KUKA KRL program: kukaSplineTemplate.src, kukaSplineTemplate.dat

--- kukaSplineTemplate.src ---
&ACCESS RVP
&REL 2
&PARAM EDITMASK = *
&PARAM TEMPLATE = C:\KRC\Roboter\Template\vorgabe
DEF mimi( )
;FOLD INI;%{PE}
  ;FOLD BASISTECH INI
    GLOBAL INTERRUPT DECL 3 WHEN $STOPMESS==TRUE DO IR_STOPM ( )
    INTERRUPT ON 3
    BAS (#INITMOV,0 )
  ;ENDFOLD (BASISTECH INI)
  ;FOLD USER INI
    ;Make your modifications here

  ;ENDFOLD (USER INI)
;ENDFOLD (INI)

;FOLD PTP HOME  Vel= 2 % DEFAULT;%{PE}%MKUKATPBASIS,%CMOVE,%VPTP,%P 1:PTP, 2:HOME, 3:, 5:100, 7:DEFAULT
$BWDSTART = FALSE
PDAT_ACT=PDEFAULT
FDAT_ACT=FHOME
BAS (#PTP_PARAMS,2 )
$H_POS=XHOME
PTP  XHOME
;ENDFOLD

$BWDSTART=FALSE
LDAT_ACT=LCPDAT[[firstIndex]]
FDAT_ACT=FP[[firstIndex]]
BAS(#CP_PARAMS,2)

;FOLD Shape SPLINE
	SPLINE
		TIME_BLOCK START
		[[range .Points]]
			SPL XP[[.Index]]
			[[if .TimeMark]]
			;Time mark at [[.TimeCode]]s with value [[.TimeMark]]s
			TIME_BLOCK PART = [[.TimeMark]]
			[[end]]
			[[if rMarkTest .Index .TimeMark]]
			;Time mark at [[.TimeCode]]s with value [[rTime]]s
			TIME_BLOCK PART = [[rTime]]
			[[end]]
		[[end]]
		TIME_BLOCK END = [[totalTime]]
	ENDSPLINE
;ENDFOLD

;FOLD WAIT Time=2.5 sec;%{PE}%R 8.3.31,%MKUKATPBASIS,%CWAIT,%VWAIT,%P 3:2.5
WAIT SEC 2.5
;ENDFOLD

;FOLD PTP HOME  Vel= 2 % DEFAULT;%{PE}%MKUKATPBASIS,%CMOVE,%VPTP,%P 1:PTP, 2:HOME, 3:, 5:100, 7:DEFAULT
$BWDSTART = FALSE
PDAT_ACT=PDEFAULT
FDAT_ACT=FHOME
BAS (#PTP_PARAMS,2 )
$H_POS=XHOME
PTP  XHOME
;ENDFOLD

END

--- kukaSplineTemplate.dat ---
&ACCESS RVP
&REL 2
&PARAM EDITMASK = *
&PARAM TEMPLATE = C:\KRC\Roboter\Template\vorgabe
DEFDAT  kimchiandchips
;FOLD EXTERNAL DECLARATIONS;%{PE}%MKUKATPBASIS,%CEXT,%VCOMMON,%P
;FOLD BASISTECH EXT;%{PE}%MKUKATPBASIS,%CEXT,%VEXT,%P
EXT  BAS (BAS_COMMAND  :IN,REAL  :IN )
DECL INT SUCCESS
;ENDFOLD (BASISTECH EXT)
;FOLD USER EXT;%{E}%MKUKATPUSER,%CEXT,%VEXT,%P
;Make your modifications here

;ENDFOLD (USER EXT)
;ENDFOLD (EXTERNAL DECLARATIONS)
DECL BASIS_SUGG_T LAST_BASIS={POINT1[] "P[[fTotal]]",POINT2[] "P[[fTotal]]",CP_PARAMS[] "CPDAT[[pTotal]]",PTP_PARAMS[] "PDAT0                   ",CONT[] "                        ",CP_VEL[] "2                     ",PTP_VEL[] "100                     ",SYNC_PARAMS[] "SYNCDAT                 ",SPL_NAME[] "S0                      ",A_PARAMS[] "ADAT0                   "}
[[range .Points]]
DECL E6POS XP[[.Index]]={X [[.X]],Y [[.Y]],Z [[.Z]],A   [[.A]],B   [[.B]],C   [[.C]],S [[.S]],T [[.T]],E1 [[.E1]],E2 [[.E2]],E3 [[.E3]],E4 [[.E4]],E5 [[.E5]],E6 [[.E6]]}
[[if first .Index]]DECL FDAT FP[[.Index]]={TOOL_NO 1,BASE_NO 0,IPO_FRAME #BASE,POINT2[] " ",TQ_STATE FALSE}
DECL LDAT LCPDAT[[.Index]]={VEL 2.00000,ACC 50.000,APO_DIST 100.000,APO_FAC 50.0000,AXIS_VEL 100.000,AXIS_ACC 25.000,ORI_TYP #VAR,CIRC_TYP #BASE,JERK_FAC 50.0000,GEAR_JERK 50.0000,EXAX_IGN 0}[[end]]
[[end]]

ENDDAT
